// TIA Portal V18 export
DATA_BLOCK "SS1_CPU1214_DO_Vars"   // DB11014
{ S7_Optimized_Access := 'FALSE' }
VERSION : 0.1
// stored: AutoNumber false, DBAccessibleFromOPCUA true, IsOnlyStoredInLoadMemory false, IsWriteProtectedInAS false
   VAR
      DO1 { S7_SetPoint := 'True'} : "UDT_DOadv";   // Резерв
      DO2 { S7_SetPoint := 'True'} : "UDT_DOadv";   // Резерв
      DO3 { S7_SetPoint := 'True'} : "UDT_DOadv";   // Резерв
      DO4 { S7_SetPoint := 'True'} : "UDT_DOadv";   // Резерв
      DO5 { S7_SetPoint := 'True'} : "UDT_DOadv";   // Резерв
      DO6 : "UDT_DOadv";   // Резерв
      DO7 { S7_SetPoint := 'True'} : "UDT_DOadv";   // Резерв
      DO8 { S7_SetPoint := 'True'} : "UDT_DOadv";   // Резерв
      DO9 { S7_SetPoint := 'True'} : "UDT_DOadv";   // Резерв
      DO10 { S7_SetPoint := 'True'} : "UDT_DOadv";   // Резерв
   END_VAR
BEGIN
END_DATA_BLOCK
